{attribute 'qualified_only'}
{attribute 'strict'}
{attribute 'to_string'}
TYPE E_DS402EGU  :
(
    MM:=0,
    UM:=1,
    NM:=2
);
END_TYPE

(* stored: Version 1.1.0.1
   DUT E_DS402EGU: Id {f02e6df6-ea84-4565-a766-82560a3f824e} *)
